PROGRAM MAIN_1_1
VAR CONSTANT
	DINT_Size:DINT :=2147483647;
	Byte_Size:DINT :=255;
END_VAR
VAR
	EP3751_0160_X AT%I*:DINT;
	EP3751_0160_Y AT%I*:DINT;
	EP3751_0160_Z AT%I*:DINT;
	
	
	EP3751_0260_X AT%I*:DINT;
	EP3751_0260_Y AT%I*:DINT;
	EP3751_0260_Z AT%I*:DINT;	
	EP3751_0260_rX AT%I*:DINT;
	EP3751_0260_rY AT%I*:DINT;
	EP3751_0260_rZ AT%I*:DINT;
	
	
	stEL6851InData  AT%I*:  ST_EL6851InDataEx;
	stEL6851OutData AT%Q*: ST_EL6851OutData;
	stCommandBuffer : ST_DMXCommandBuffer;
	arrProcessData  : ARRAY [1..512] OF BYTE;
	
	fbDMX		: FB_EL6851CommunicationEx;
	fbSample	: TON;
	bEP3751_0160_active AT%I*:BOOL;
	aButtons	AT%I*: ARRAY [1..4] OF   BOOL;
	aLeds		AT%Q*: ARRAY [1..8] OF   BOOL;
	aTrig		: array[1..4] of r_trig;
	nIndex: INT;
	nState: INT:=2;
END_VAR

FOR nIndex:=1 TO 4 DO
	aTrig[nIndex](clk:=aButtons[nIndex]);
	IF aTrig[nIndex].Q  THEN
		IF  nState=nIndex THEN
			nState:=0; 
		ELSE
			nState:=nIndex;
		END_IF
	END_IF
END_FOR		

Memset(ADR(aLeds),0, SIZEOF(aLeds));

CASE nState OF 
	0: 	//No Control
		arrProcessData[1]:=0;
		arrProcessData[2]:=0;
		arrProcessData[3]:=0;
		arrProcessData[4]:=0;
		arrProcessData[5]:=0;
		arrProcessData[6]:=0;
		
	1: // Box without Gyro
		aLeds[1]:=TRUE;
		arrProcessData[1]:=TO_BYTE(LIMIT(0,(EP3751_0160_X*128/1100)+128,255));
		arrProcessData[2]:=TO_BYTE(LIMIT(0,(EP3751_0160_Y*128/1100)+128,255));
		arrProcessData[3]:=25;
		arrProcessData[5]:=255;
		arrProcessData[6]:=10;
		
		(*arrProcessData[1]:=TO_BYTE(LIMIT(0,(EP3751_0160_X*128/1100)+128,255));
		arrProcessData[2]:=TO_BYTE(LIMIT(0,(EP3751_0160_Y*128/1100)+128,255));
		arrProcessData[3]:=0;
		arrProcessData[5]:=0;
		arrProcessData[6]:=0;*)
		//arrProcessData[3]:=TO_BYTE((EP3751_0160_Z/DINT_Size)*256+128);
		//arrProcessData[1]:=LIMIT(0,TO_BYTE(arrProcessData[1]+(EP3751_0160_X/DINT_Size)),255);
		//arrProcessData[2]:=LIMIT(0,TO_BYTE(arrProcessData[2]+(EP3751_0160_Y/DINT_Size)),255);
		//arrProcessData[3]:=LIMIT(0,TO_BYTE(arrProcessData[3]+(EP3751_0160_Z/DINT_Size)),255);
		//arrProcessData[4]:=255;	
		
	2: // Box with Gyro
		aLeds[2]:=TRUE;
		arrProcessData[1]:=TO_BYTE(LIMIT(0,(EP3751_0160_X*128/1100)+128,255));
		arrProcessData[2]:=TO_BYTE(LIMIT(0,(EP3751_0160_Y*128/1100)+128,255));
		arrProcessData[3]:=10;
		arrProcessData[5]:=255;
		arrProcessData[6]:=10;
		
	3: // Box without Gyro and Color
		aLeds[3]:=TRUE;
		arrProcessData[1]:=TO_BYTE(LIMIT(0,(EP3751_0160_X*128/1100)+128,255));
		arrProcessData[2]:=TO_BYTE(LIMIT(0,(EP3751_0160_Y*128/1100)+128,255));
		arrProcessData[3]:=30;
		arrProcessData[5]:=255;
		arrProcessData[6]:=10;
		
	4: // Box with Gyro and Color
		aLeds[4]:=TRUE;
		arrProcessData[1]:=0;
		arrProcessData[2]:=0;
		arrProcessData[3]:=0;
		arrProcessData[4]:=0;
		arrProcessData[5]:=0;
		arrProcessData[6]:=0;
END_CASE


fbDMX(
	wSourceManufacturerId:= 16#42_41, 
	dwSourceDeviceId:= 16#12_13_14_15, 
	bEnableSendingData:= TRUE, 
	bSetCycleMode:=TRUE , 
	bSendDefaultData:= , 
	uiDataLength:= 64 , 
	dwOptions:=  , 
	stEL6851InData:=	stEL6851InData , 
	stEL6851OutData:= 	stEL6851OutData, 
	stCommandBuffer:= 	stCommandBuffer, 
	arrProcessData:=	arrProcessData);

END_PROGRAM

(* stored: Version 1.1.0.1, ProductVersion 3.1.4024.12
   POU MAIN_1_1: Id {a5cd325d-529c-4168-8fae-36ca7db0453f}, SpecialFunc None *)
